// TwinCAT 3 PLC project PLC_Regression
// ProgramVersion: 3.1.4024.0
// libraries:
//   Tc2_Standard, * (Beckhoff Automation GmbH)
//   Tc2_System, * (Beckhoff Automation GmbH)
//   Tc3_Module, * (Beckhoff Automation GmbH)
//   Tc3_Vision, * (Beckhoff Automation GmbH)
// project tree:
//   DUTs/ ESvmRegressorType.TcDUT, E_RegressorType.TcDUT, ST_RegressorParams.TcDUT
//   / PlcTask.TcTTO
//   POUs/ FB_TrainingDataHandler.TcPOU, F_ExtractFeatures.TcPOU, MAIN.TcPOU
// real-time tasks:
//   TASK PlcTask: cycle T#10ms, priority 20, ADS port 350
//   TASK VnTask ImgAcq (TrainingImages): cycle T#10ms, priority 5, ADS port 351
//   TASK VnTask ImgAcq (TestImages): cycle T#10ms, priority 6, ADS port 352

CONFIGURATION PLC_Regression
    RESOURCE PLC ON TwinCAT3
        TASK PlcTask(INTERVAL := T#10ms, PRIORITY := 20);
        PROGRAM MAIN WITH PlcTask : MAIN;
    END_RESOURCE
END_CONFIGURATION

// ---- DUTs/ESvmRegressorType.TcDUT
{attribute 'qualified_only'}
{attribute 'strict'}
TYPE ESvmRegressorType :
(
	EPS := TO_UDINT(ETcVnSvm.TCVN_SVM_EPS_REGRESSOR),
	NU := TO_UDINT(ETcVnSvm.TCVN_SVM_NU_REGRESSOR)
) UDINT;
END_TYPE

// ---- DUTs/E_RegressorType.TcDUT
{attribute 'qualified_only'}
{attribute 'strict'}
TYPE E_RegressorType :
(
	KNN := 0,
	RTrees,
	STA,
	SVM
);
END_TYPE

// ---- DUTs/ST_RegressorParams.TcDUT
TYPE ST_RegressorParams :
STRUCT
	nKnnK							:	UDINT 				:=	2;
	nRTreesMaxDepth					:	UDINT				:=	5;			// optional Exp parameter
	nRTreesMinSamples				:	UDINT				:=	2;			// optional Exp parameter
	nRTreesActiveVariables			:	UDINT				:=	0;			// optional Exp parameter
	nRTreesMaxIterations			:	UDINT				:=	50;			// optional Exp parameter
	fRTreesEpsilon					:	LREAL				:=	0.1;		// optional Exp parameter
	fRTreesRegressionAccuracy		:	REAL				:=	0.0;		// optional Exp parameter
	fStaRho	                        :	LREAL				:=	0.99;
	nStaNu	                        :	UDINT				:=	5;			// optional Exp parameter
	bStaDoublePrecision				:	BOOL				:=	TRUE;		// optional Exp parameter
	fStaBetaSbm						:	LREAL				:=	0.0;		// optional Exp parameter
	nStaPhi							:	UDINT				:=	1;			// optional Exp parameter
	nStaTau							:	UDINT				:=	100;		// optional Exp parameter
	eSvmType						:	ESvmRegressorType	:=	ESvmRegressorType.EPS;
	fSvmC							:	LREAL				:=	1000;
	fSvmNu							:	LREAL				:=	0.2;
	fSvmP							:	LREAL				:=	1;
	eSvmKernelType					:	ETcVnSvmKernelType	:=	ETcVnSvmKernelType.TCVN_SKT_RBF;
	fSvmGamma						:	LREAL				:=	1;
	fSvmCoef0						:	LREAL				:=	0;
	fSvmDegree						:	LREAL				:=	0;
	nSvmMaxIterations				:	UDINT				:=	100000;		// optional Exp parameter
	fSvmEpsilon						:	LREAL				:=	0.00001;	// optional Exp parameter
END_STRUCT
END_TYPE

// ---- POUs/MAIN.TcPOU
PROGRAM MAIN
VAR
	eRegressorType		: 	E_RegressorType;		// Regressor type
	stParams			:	ST_RegressorParams;		// Regressor parameters
	bResetModel			:	BOOL;					// Reset model to start a new training with a changed model or parameters
	bResetTrainingData	:	BOOL;					// Reset the trained features to get new ones and train model
	eTrainedModelType	: 	E_RegressorType;
	
	hrTrain				:	HRESULT;
	hrTest				:	HRESULT;
	
	ipImageTest			:	ITcVnImage;
	ipImageResDisp		:	ITcVnDisplayableImage;
	
	eCameraState		:	ETcVnCameraState;	
	fbCameraTest		:	FB_VN_SimpleCameraControl;
	
	fbTrainingDataHandler:	FB_TrainingDataHandler;
	
	ipRegressorModel	:	ITcVnMlModel;
	ipSamplesTraining	:	ITcVnContainer;
	ipScalarTargets		:	ITcVnContainer;
	ipFeatureScaling	:	ITcVnContainer;
	ipSampleTest		:	ITcVnContainer;
	ipStaPredictionScaling:	ITcVnContainer;
	fPredictedScalar	:	REAL;
	fNovelty			:	REAL;
	
	// Result
	fNoveltyThreshold	:	REAL;
	sLabel				:	STRING(255);
	aGreen				:	TcVnVector4_LREAL := [0, 255, 0];
END_VAR

// Disclaimer

// This publication contains statements about the suitability of our products for certain
// areas of application. These statements are based on typical features of our products.
// The examples shown in this publication are for demonstration purposes only.
// The information provided herein should not be regarded as specific operation characteristics.
// It is incumbent on the customer to check and decide whether a product is suitable for use
// in a particular application. We do not give any warranty that the source code which is
// made available with this publication is complete or accurate.

// THE SAMPLE CODE CONTAINED IN THIS PUBLICATION IS PROVIDED “AS IS” WITHOUT WARRANTY OF ANY KIND,
// EITHER EXPRESSED, IMPLIED OR STATUTORY, INCLUDING WITHOUT LIMITATION, ANY WARRANTY WITH RESPECT TO NON-INFRINGEMENT,
// FREEDOM FROM PROPRIETARY RIGHTS OF THIRD PARTIES OR FITNESS FOR ANY PARTICULAR PURPOSE.

// This publication may be changed from time to time without prior notice.
// No liability is assumed for errors and/or omissions.
// Our products are described in detail in our data sheets and documentations.
// Product-specific warnings and cautions must be observed.
// For the latest version of our data sheets and documentations visit our website (www.beckhoff.de).

// © Beckhoff Automation GmbH & Co. KG, December 2023

// The reproduction, distribution and utilization of this document as well as the communication
// of its contents to others without express authorization is prohibited. 
// Offenders will be held liable for the payment of damages.
// All rights reserved in the event of the grant of a patent, utility model or design.

//	==========================================================================================

// SAMPLE - Machine Learning Regression
//	-------------------------------------------------------

// Steps To Do:
// ------------
// 1. Add the training images to the TrainingImages control
// 2. Add the test images to the TestingImages control
// 3. Activate the configuration -> Start TwinCAT system and PLC to run -> watch the results in the ADS Image Watch
// 4. Change eRegressorType and stParams to change the model or settings
// 5. Set bResetModel to start create a new model and start training
//    Note: If you change to eClassifierType = STA or from this type to another, a bResetTrainingData is automatically performed due to the different scaling of the training data.
// 6. Set bResetTrainingData to get new training data if images or feature extraction changed

// Reset the trained features to get new ones and train model
IF bResetTrainingData
	OR (eTrainedModelType <> E_RegressorType.STA AND eRegressorType = E_RegressorType.STA) 
	OR (eTrainedModelType = E_RegressorType.STA AND eRegressorType <> E_RegressorType.STA) THEN
	
	bResetTrainingData := FALSE;
	fbTrainingDataHandler.Reset();
	FW_SafeRelease(ADR(ipSamplesTraining));
	FW_SafeRelease(ADR(ipScalarTargets));
	FW_SafeRelease(ADR(ipFeatureScaling));
	FW_SafeRelease(ADR(ipRegressorModel));
	FW_SafeRelease(ADR(ipStaPredictionScaling));
	eTrainedModelType := eRegressorType;
	// Reset return value
	hrTrain := S_OK;
END_IF

// Get sample data for training
fbTrainingDataHandler(eRegressorType := eRegressorType);
IF ipSamplesTraining = 0 AND ipScalarTargets = 0 AND ipFeatureScaling = 0 AND ipStaPredictionScaling = 0 THEN
	hrTrain := fbTrainingDataHandler.GetTrainingData(ipSamplesTraining, ipScalarTargets, ipStaPredictionScaling, ipFeatureScaling);
END_IF

// Retrain with changed model or parameters
IF bResetModel THEN
	bResetModel := FALSE;
	FW_SafeRelease(ADR(ipRegressorModel));
	eTrainedModelType := eRegressorType;
	// Reset return value
	hrTrain := S_OK;
END_IF

IF SUCCEEDED(hrTrain) AND ipSamplesTraining <> 0 AND ipScalarTargets <> 0 AND ipRegressorModel = 0 THEN
	
	// Create the model
	CASE eRegressorType OF
		
		E_RegressorType.KNN:
			hrTrain := F_VN_CreateKnnModel(
								ipMlModel			:=	ipRegressorModel,
								eKnnType			:=	TCVN_KNN_REGRESSOR,
								nK					:=	stParams.nKnnK,
								hrPrev				:=	hrTrain);
			
			// Set novelty threshold according to model results
			fNoveltyThreshold := 0.1;
			
		E_RegressorType.RTrees:
			hrTrain := F_VN_CreateRTreesModelExp2(
								ipMlModel			:=	ipRegressorModel,
								eRTreesType			:=	TCVN_RT_REGRESSOR,
								nMaxDepth			:=	stParams.nRTreesMaxDepth,
								nMinSamples			:=	stParams.nRTreesMinSamples,
								nActiveVariables	:=	stParams.nRTreesActiveVariables,
								nMaxiterations		:=	stParams.nRTreesMaxIterations,
								fEpsilon			:=	stParams.fRTreesEpsilon,
								fRegressionAccuracy	:=	stParams.fRTreesRegressionAccuracy,
								ipClassPriors		:=	0,
								hrPrev				:=	hrTrain);

		E_RegressorType.STA:
			hrTrain := F_VN_CreateStaModelExp2(
								ipMlModel           :=	ipRegressorModel,
								eStaType            :=	TCVN_STA_REGRESSOR,
								fRho                :=	stParams.fStaRho,
								nNu                 :=	stParams.nStaNu,
								bDoublePrecision    :=	stParams.bStaDoublePrecision,
								fBetaSbm			:=	stParams.fStaBetaSbm, 
								nPhi				:=	stParams.nStaPhi, 
								nTau				:=	stParams.nStaTau, 
								hrPrev				:=	hrTrain); 

			// Set novelty threshold according to model results
			fNoveltyThreshold := 0.2;
			
		E_RegressorType.SVM:
			hrTrain := F_VN_CreateSvmModelExp(
								ipMlModel			:=	ipRegressorModel,
								eSvmType			:=	TO_UDINT(stParams.eSvmType),
								fC					:=	stParams.fSvmC,
								fNu					:=	stParams.fSvmNu,
								fP					:=	stParams.fSvmP,
								eKernelType			:=	stParams.eSvmKernelType,
								fGamma				:=	stParams.fSvmGamma,
								fCoef0				:=	stParams.fSvmCoef0,
								fDegree				:=	stParams.fSvmDegree,
								nMaxIterations		:=	stParams.nSvmMaxIterations,
								fEpsilon			:=	stParams.fSvmEpsilon,
								hrPrev				:=	hrTrain);
	
	END_CASE
	
	// Train model
	hrTrain := F_VN_TrainBatch(
					ipMlModel   :=  ipRegressorModel,
					ipSamples   :=  ipSamplesTraining,
					ipOutputs   :=  ipScalarTargets,
					hrPrev      :=  hrTrain);

END_IF

// Get test images
eCameraState := fbCameraTest.GetState();

IF eCameraState = TCVN_CS_ERROR THEN
	hrTest := fbCameraTest.Reset();

ELSIF eCameraState < TCVN_CS_ACQUIRING THEN
	hrTest := fbCameraTest.StartAcquisition();

// Camera streaming
ELSIF eCameraState = TCVN_CS_ACQUIRING THEN
	hrTest := fbCameraTest.GetCurrentImage(ipImageTest);

	// Check if new image was received
	IF SUCCEEDED(hrTest) AND ipImageTest <> 0 THEN

        IF ipRegressorModel <> 0 AND ipFeatureScaling <> 0 THEN
			// Get features from sample image and scale 
			hrTest := F_ExtractFeatures(ipImageTest, ipSampleTest, hrTest);
			IF eRegressorType = E_RegressorType.STA THEN
				hrTest := F_VN_FeatureScalingExp(ipSampleTest, ipFeatureScaling, ipSampleTest, 0.1, 0.9, hrTest);
			ELSE
				hrTest := F_VN_FeatureScaling(ipSampleTest, ipFeatureScaling, ipSampleTest, hrTest);
			END_IF
			
			// Prediction with optional novelty calculation if supported
			CASE eRegressorType OF
			
				E_RegressorType.KNN, E_RegressorType.STA:
					// Predict scalar result and novelty
					hrTest := F_VN_PredictSampleScalarExp(ipRegressorModel, ipSampleTest, fPredictedScalar, fNovelty, hrTest);
					
					IF eRegressorType = E_RegressorType.STA AND ipStaPredictionScaling <> 0 THEN
						// Inverse scaling of the prediction result to get the original target value range
						hrTest := F_VN_InverseFeatureScalingExp_REAL(fPredictedScalar, ipStaPredictionScaling, fPredictedScalar, 0.1, 0.9, hrTest);
					END_IF
				
					// Check the degree of novelty and get result
					IF fNovelty <= fNoveltyThreshold THEN
						sLabel := CONCAT('Prediction: ',REAL_TO_STRING(fPredictedScalar));
					ELSE
						sLabel := 'Prediction: Unknown';
					END_IF
			ELSE
				// Predict scalar result
				hrTest := F_VN_PredictSampleScalar(ipRegressorModel, ipSampleTest, fPredictedScalar, hrTest);
				// Get result
				sLabel := CONCAT('Prediction: ',REAL_TO_STRING(fPredictedScalar));				
			END_CASE
			
			// Write result
			hrTest := F_VN_PutTextExp(sLabel, ipImageTest, 22, 70, TCVN_FT_HERSHEY_PLAIN, 3, aGreen, 2, TCVN_LT_ANTIALIASED, FALSE, hrTest);
		END_IF
		
		// Display Image
		hrTest := F_VN_TransformIntoDisplayableImage(ipImageTest, ipImageResDisp, S_OK);
	END_IF
END_IF

END_PROGRAM

// ---- POUs/FB_TrainingDataHandler.TcPOU
FUNCTION_BLOCK PUBLIC FB_TrainingDataHandler
VAR_INPUT
	eRegressorType 		: E_RegressorType;	
END_VAR
VAR_OUTPUT
END_VAR
VAR
	hr					: HRESULT;
	eCameraState		: ETcVnCameraState;
	fbCameraTraining	: FB_VN_SimpleCameraControl;	
	ipImageTraining		: ITcVnImage;
	ipImageTrainingDisp	: ITcVnDisplayableImage;
	bTrigger			: BOOL := TRUE;
	sLabel				: STRING(255);
	aGreen				: TcVnVector4_LREAL := [0, 255, 0];
	
	// Image Info
	nImagesTotal		: UDINT := 22;
	nImagesLoaded		: UDINT := 0;
	
	ipFeatures			: ITcVnContainer;
	ipImageFeatures		: ITcVnContainer;
	ipLabels			: ITcVnContainer;
	ipStaResultScaling	: ITcVnContainer;
	ipScales			: ITcVnContainer;
	ipScaledFeatures	: ITcVnContainer;
	
	// The measured distance between the camera and the object in each image in cm
	aGroundTruth		: ARRAY [0..21] OF LREAL := [17, 19, 21, 23, 25, 27, 29, 31, 33, 35, 37, 39, 41, 43, 45, 47, 49, 51, 53, 55, 57, 59];
END_VAR

// Initialize container
IF ipImageFeatures = 0 THEN
	hr := F_VN_CreateContainer(ipImageFeatures, ContainerType_Vector_Vector_LREAL, nImagesTotal, hr);
	hr := F_VN_CreateContainerFromArray(ADR(aGroundTruth), ipLabels, ContainerType_Vector_LREAL, 22, hr);
END_IF

// Get training images
eCameraState := fbCameraTraining.GetState();

IF eCameraState = TCVN_CS_ERROR THEN
	hr := fbCameraTraining.Reset();
	
// Camera trigger image
ELSIF eCameraState = TCVN_CS_TRIGGERING THEN
	hr := fbCameraTraining.TriggerImage();
	
ELSIF eCameraState < TCVN_CS_ACQUIRING THEN
	hr := fbCameraTraining.StartAcquisition();

// Camera streaming
ELSIF eCameraState = TCVN_CS_ACQUIRING THEN

	IF bTrigger THEN
		hr := fbCameraTraining.TriggerImage();
		IF SUCCEEDED(hr) THEN
			bTrigger := FALSE;
		END_IF
	ELSE
		hr := fbCameraTraining.GetCurrentImage(ipImageTraining);

		// Check if new image was received
		IF SUCCEEDED(hr) AND ipImageTraining <> 0 THEN
			
			// Get features from training image 
			hr := F_ExtractFeatures(ipImageTraining, ipFeatures, hr);
			
			// Add features to the container
			hr := F_VN_SetAt_ITcVnContainer(ipFeatures, ipImageFeatures, nImagesLoaded, hr);
			FW_SafeRelease(ADR(ipFeatures));
			
			// Display image
			sLabel := CONCAT('Image Number: ', UDINT_TO_STRING(nImagesLoaded + 1));
			hr := F_VN_PutTextExp(sLabel, ipImageTraining, 50, 100, TCVN_FT_HERSHEY_PLAIN, 3, aGreen, 2, TCVN_LT_ANTIALIASED, FALSE, hr);
			hr := F_VN_TransformIntoDisplayableImage(ipImageTraining, ipImageTrainingDisp, hr);
			
			nImagesLoaded := nImagesLoaded + 1;
			IF nImagesLoaded < nImagesTotal THEN
				// Trigger next image
				bTrigger := TRUE;
			ELSE
				// After collecting all training data, normalize the feature values
				hr := F_VN_GetFeatureScales(ipImageFeatures, ipScales, TCVN_FST1_MINMAX, hr);
				IF eRegressorType = E_RegressorType.STA THEN
					hr := F_VN_FeatureScalingExp(ipImageFeatures, ipScales, ipScaledFeatures, 0.1, 0.9, hr);
					hr := F_VN_GetFeatureScales(ipLabels, ipStaResultScaling, TCVN_FST1_MINMAX, hr);
					hr := F_VN_FeatureScalingExp(ipLabels, ipStaResultScaling, ipLabels, 0.1, 0.9, hr);
				ELSE
					hr := F_VN_FeatureScaling(ipImageFeatures, ipScales, ipScaledFeatures, hr);
					FW_SafeRelease(ADR(ipStaResultScaling));
				END_IF
				FW_SafeRelease(ADR(ipImageFeatures));
			END_IF
		END_IF
	END_IF
END_IF

METHOD PUBLIC GetTrainingData : HRESULT
VAR_INPUT
	ipTrainingSamples		: REFERENCE TO ITcVnContainer;
	ipClassLabels			: REFERENCE TO ITcVnContainer;
	ipStaPredictionScaling	: REFERENCE TO ITcVnContainer;
	ipFeatureScaling		: REFERENCE TO ITcVnContainer;
END_VAR
VAR
	hr						: HRESULT;
END_VAR
IF nImagesLoaded = nImagesTotal THEN
	hr := F_VN_CopyContainer(ipScaledFeatures, ipTrainingSamples, hr);
	hr := F_VN_CopyContainer(ipLabels, ipClassLabels, hr);
	IF eRegressorType = E_RegressorType.STA THEN
		hr := F_VN_CopyContainer(ipStaResultScaling, ipStaPredictionScaling, hr);
	END_IF
	GetTrainingData := F_VN_CopyContainer(ipScales, ipFeatureScaling, hr);
ELSE
	GetTrainingData := S_PENDING;
END_IF
END_METHOD

METHOD PUBLIC Reset : HRESULT
VAR_INPUT
END_VAR
nImagesLoaded := 0;
FW_SafeRelease(ADR(ipFeatures));
FW_SafeRelease(ADR(ipImageFeatures));
FW_SafeRelease(ADR(ipLabels));
FW_SafeRelease(ADR(ipStaResultScaling));
FW_SafeRelease(ADR(ipScales));
FW_SafeRelease(ADR(ipScaledFeatures));
bTrigger := TRUE;
END_METHOD

END_FUNCTION_BLOCK

// ---- POUs/F_ExtractFeatures.TcPOU
FUNCTION F_ExtractFeatures : HRESULT
VAR_INPUT
	ipImage			:	ITcVnImage;
	ipFeatures		:	REFERENCE TO ITcVnContainer;
	hrPrev			:	HRESULT;
END_VAR
VAR
	hr				:	HRESULT;
	stPixelFormat	:	TcVnPixelFormat;
	ipImageWork 	:	ITcVnImage;
	ipContourList	:	ITcVnContainer;
	ipIterator		:	ITcVnForwardIterator;
	ipContour		:	ITcVnContainer;
	fArea			:	LREAL;
	fMaxArea		:	LREAL;
	aCenter			:	TcVnPoint2_REAL;
	fRadius			:	REAL;
	aFeatures		:	ARRAY [0..1] OF LREAL;
END_VAR

IF FAILED(hrPrev) THEN
	F_ExtractFeatures := hrPrev;
	RETURN;
END_IF

IF ipImage = 0 THEN
	F_ExtractFeatures := Tc2_System.E_HRESULTAdsErr.INVALIDPARM;
	RETURN;
END_IF

// Convert image from RGB to Gray if nessesary
hr := F_VN_GetPixelFormat(ipImage, stPixelFormat, hr); 
IF stPixelFormat.nChannels = 3 AND stPixelFormat.ePixelEncoding = TCVN_PE_NONE THEN
	hr := F_VN_ConvertColorSpace(ipImage, ipImageWork, TCVN_CST_RGB_TO_GRAY, hr);
ELSE
	ipImageWork := ipImage;
	ipImage.TcAddRef();
END_IF
		
// Simple feature extraction example
hr := F_VN_Threshold(ipImageWork, ipImageWork, 220, 255, TCVN_TT_BINARY_INV, hr);
hr := F_VN_FindContours(ipImageWork, ipContourList, hr);

// Find the largest contour in the image
hr := F_VN_GetForwardIterator(ipContourList, ipIterator, hr);
WHILE SUCCEEDED(hr) AND_THEN ipIterator.CheckIfEnd() <> S_OK DO
	hr := F_VN_GetContainerExp(ipIterator, ipContour, 1, hr);

	hr := F_VN_ContourArea(ipContour, fArea, hr);
	IF fArea > fMaxArea THEN
		// Extract the features of the contour
		aFeatures[0] := fMaxArea := fArea;
		hr := F_VN_EnclosingCircle(ipContour, aCenter, fRadius, hr);
		aFeatures[1] := REAL_TO_LREAL(fRadius);
	END_IF
END_WHILE

// Create a container with all features as a vector
hr := F_VN_CreateContainerFromArray(ADR(aFeatures), ipFeatures, ContainerType_Vector_LREAL, 2, hr);

// Release interface pointer
FW_SafeRelease(ADR(ipImageWork));
FW_SafeRelease(ADR(ipContourList));
FW_SafeRelease(ADR(ipIterator));
FW_SafeRelease(ADR(ipContour));

F_ExtractFeatures := hr;

END_FUNCTION
